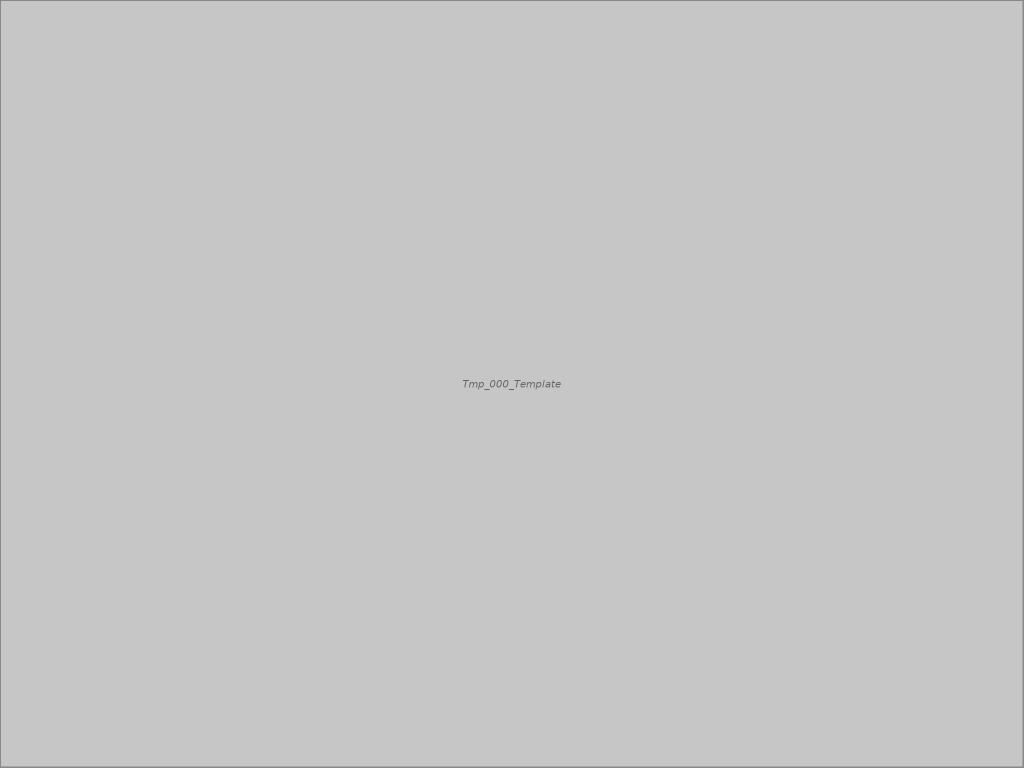
VISUALIZATION Lay_040_MachineLayout  // 1024x768
    Frame (0,0 1024x768)
        shows Tmp_000_Template(header := gHMIData.hmiHeader)
END_VISUALIZATION

(* stored: Version 1.1.0.1, ProductVersion 3.1.4024.11
   Visu Lay_040_MachineLayout: Id {88ee6430-3b99-476f-997c-dbe82955d6be} *)
